FUNCTION_BLOCK Room_Ctx_Hmi
VAR_INPUT
	sStatusText				: Str;
	sErrorText				: Str;
	nStatusColor			: LWORD;
	
	bDisable				: BOOL;	
END_VAR
VAR_OUTPUT PERSISTENT
	nTimeout				: UDINT := TIME_TO_UDINT(T#60S);	

	rMaxTemperature			: REAL := 19.5; // °C
	rMinTemperature			: REAL := 19.0; // °C
END_VAR

END_FUNCTION_BLOCK

(* stored: Version 1.1.0.1
   POU Room_Ctx_Hmi: Id {9536c277-9786-455b-b876-b447754e1a8d}, SpecialFunc None *)
